(* CoDeSys 2.3.9.42 project: PROYECTO_FINAL.pro *)
(* Libraries: Standard.LIB 4.10.05 12:14:46, Iecsfc.lib 13.4.06 15:51:28 *)

(* Global variable list: Global_Variables *)
VAR_GLOBAL


(*ENTRADAS*)

	M:BOOL;(*Boton para iniciar el proceso automatico*)
	Marcha:BOOL;(*Variable que se pone a 1 cuando apretamos M*)
	Auto:BOOL;(*Cambio de modo automatico a manual*)


	P:BOOL;(*Boton para parar el proceso automatico*)
	E:BOOL;(*Boton para iniciar el proceso de emergencia*)
	Rearme:BOOL;(*Boton para reiniciar el proceso*)

	Mesa1:BOOL;(*Boton para Mesa 1*)
	Mesa2:BOOL;(*Boton para Mesa 2*)
	Mesa3:BOOL;(*Boton para Mesa 3*)
	Mesa4:BOOL;(*Boton para Mesa 4*)


	Pizza1:BOOL;(*Boton pizza 1: Tomate y queso*)
	Pizza2:BOOL;(*Boton pizza 2: Tomate, queso y jamon*)
	Pizza3:BOOL;(*Boton pizza 3:Tomate,queso y peperoni*)
	Pizza4:BOOL;(*Boton pizza 4:Tomate, queso, pimientos y champiñones*)
	P1:BOOL;(*Variable que se pone a 1 cuando se elige la pizza 1 y que se pone a 0 cuando se entra en el horno*)
	P2:BOOL;(*Variable que se pone a 1 cuando se elige la pizza 2 y que se pone a 0 cuando se entra en el horno*)
	P3:BOOL;(*Variable que se pone a 1 cuando se elige la pizza 3 y que se pone a 0 cuando se entra en el horno*)
	P4:BOOL;(*Variable que se pone a 1 cuando se elige la pizza 4 y que se pone a 0 cuando se entra en el horno*)


	SMasa:BOOL;(*Sensor de que la masa cae en la cinta*)
	SAmasador:BOOL;(*Sensor de que la masa esta en el punto de amasar*)

	(*Sensores ingredientes*)
	SPizza:BOOL;(*Sensor para ver que pizza se ha elegido*)
	STOM:BOOL;(*Sensor que la pizza esta en la posicion para echar tomate*)
	SQUE:BOOL;(*Sensor que la pizza esta en la posicion para echar queso*)
	SJAM:BOOL;(*Sensor que la pizza esta en la posicion para echar jamon*)
	SPEP: BOOL;(*Sensor que la pizza esta en la posicion para echar peperoni*)
	SPIM: BOOL;(*Sensor que la pizza esta en la posicion para echar pimiento*)
	SCHAMP: BOOL;(*Sensor que la pizza esta en la posicion para echar champiñones*)
	SHORNO: BOOL;(*Sensor que se activa cuando la pizza llega al horno*)
	SCarrito:BOOL;(*Sensor que se activa cuando hay un carrito en la salida del horno*)
	SMesa1:BOOL;(*Sensor que se activa cuando carrito llega a mesa 1*)
	SMesa2:BOOL;(*Sensor que se activa cuando carrito llega a mesa 2*)
	SMesa3:BOOL;(*Sensor que se activa cuando carrito llega a mesa 3*)
	SMesa4:BOOL;(*Sensor que se activa cuando carrito llega a mesa 4*)

	SEHorno:BOOL;(*Sensor de entrada horno*)
	SFHorno:BOOL;(*Sensor salida horno*)
	INVISIBLE:BOOL;(*Se activa para hacer invisible la masa*)

	(*Botones del modo Manual*)
	MAS:BOOL;(*Boton para tirar una masa a la cinta*)
	MOT:BOOL;(*Boton que activa la cinta*)
	AM:BOOL;(*Boton de amasar*)
	TOM:BOOL;(*Boton del tomate*)
	QUE:BOOL;(*Boton del queso*)
	JAM:BOOL;(*Boton del jamon*)
	PEP:BOOL;(*Boton del peperoni*)
	PIM:BOOL;(*Boton del pimiento*)
	CH:BOOL;(*Boton de los champiñones*)
	H:BOOL;(*Boton del horno*)

	(*posicion carrito*)
	PosYR:INT;(*Coordenada Y carrito*)
	PosXR:INT;(*Coordenada X carrito*)
	ActMesa1: BOOL;(*variable que se activa al elegir la mesa 1*)
	ActMesa2: BOOL;(*variable que se activa al elegir la mesa 2*)
	ActMesa3: BOOL;(*variable que se activa al elegir la mesa 3*)
	ActMesa4: BOOL;(*variable que se activa al elegir la mesa 4*)
	CargaRojo: BOOL;(*Variable para mostrar que la pizza se ha cargado en el carrito*)
	(*posicion masa*)
	PosXM:INT;
	PosYM:INT;
	AUXMasa:BOOL;(*variable auxiliar que se activa mientras la masa cae en la cinta*)





(*SALIDAS*)

	(*Acciones de la cinta*)
	Masa:BOOL;(*Accion de tirar la masa en la cinta*)
	Amasador:BOOL;(*Accion de amasar la masa*)
	Motor:BOOL;(*Motor de la cinta*)
	Horno:BOOL;(*Horno encendido*)

	(*Acciones ingredientes*)
	MT:BOOL;(*Abrir compuerta del tomate*)
	MQ:BOOL;(*Abrir compuerta del queso*)
	MJ:BOOL;(*Abrir compuerta del jamon*)
	MPE:BOOL;(*Abrir compuerta del peperoni*)
	MPI:BOOL;(*Abrir compuerta del pimiento*)
	MCH:BOOL;(*Abrir compuerta de los champiñones*)


	Vel:INT:=2;(*Velocidad para las animaciones*)






END_VAR

(* POU PLC_PRG, ST *)
PROGRAM PLC_PRG

VAR

END_VAR
Cinta;
Control;
Cambio_Modo;
Amasadora;
ControlCarritoRojo;
END_PROGRAM

(* POU CINTA_TRANSPORTADORA/Cinta, ST *)
PROGRAM Cinta
VAR

END_VAR
SMasa:=FALSE;
	SAmasador:=FALSE;
	SPizza:=FALSE;
	STOM:=FALSE;
	SQUE:=FALSE;
	SJAM:=FALSE;
	SPEP:=FALSE;
	SPIM:=FALSE;
	SCHAMP:=FALSE;
	SHORNO:=FALSE;
	SEHORNO:=FALSE;
	SFHORNO:=FALSE;

IF PosYM>=0 AND PosYM<=80 AND PosXM=0 THEN
AUXMasa:=TRUE;
END_IF


IF Masa=TRUE THEN
	PosYM:=PosYM+Vel;

END_IF

IF Motor=TRUE  THEN
	 PosXM:=PosXM+Vel;
END_IF





IF PosYM>=80AND PosXM >=0 AND PosXM<=30 THEN
	SMasa:=TRUE;
	END_IF
IF PosXM >=80 AND PosXM<=120 THEN
 SAmasador:=TRUE;
	END_IF
IF PosXM>=200 AND PosXM<=240 THEN
 SPizza:=TRUE;
	END_IF
IF PosXM >=300 AND PosXM<=340 THEN
 STOM:=TRUE;
	END_IF
IF PosXM>=370 AND PosXM<=390 THEN
 SQUE:=TRUE;
	END_IF
IF PosXM >=440 AND PosXM<=460 THEN
 SJAM:=TRUE;
	END_IF
IF PosXM >=510 AND PosXM<=530 THEN
 SPEP:=TRUE;
	END_IF
IF PosXM >=580 AND PosXM<=600 THEN
 SPIM:=TRUE;
	END_IF
IF PosXM >=650 AND PosXM<=670 THEN
 SCHAMP:=TRUE;
	END_IF
IF PosXM >=720 AND PosXM<=750 THEN
 SEHORNO:=TRUE;
	END_IF
IF PosXM >=820 AND PosXM<=840 THEN
 SFHORNO:=TRUE;
	END_IF
IF INVISIBLE=TRUE THEN
PosXM:=0;
PosYM:=0;
INVISIBLE:=FALSE;
END_IF

IF SMasa=TRUE THEN
AUXMasa:=FALSE;
END_IF
END_PROGRAM

(* POU CONTROL_AUTO/MAN/Control, SFC *)
PROGRAM Control
VAR
	OK:BOOL;
END_VAR
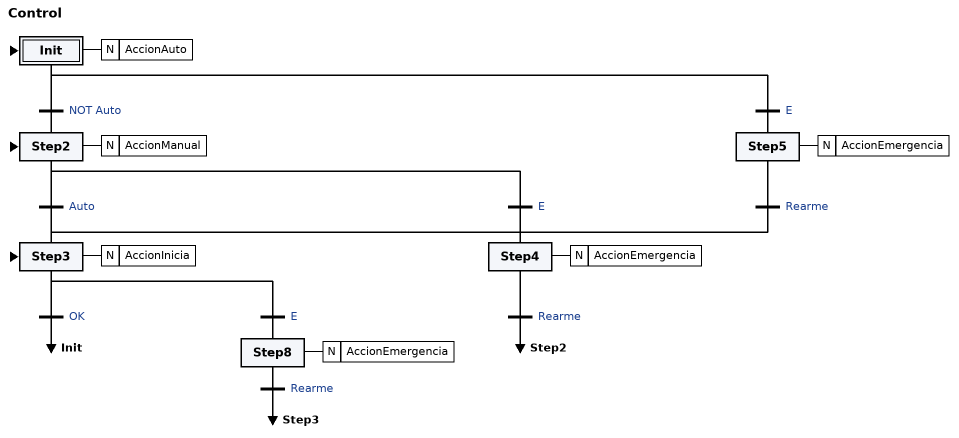
INITIAL_STEP Init:
	AccionAuto(N);
END_STEP
TRANSITION FROM Init TO Step2 := NOT Auto;
END_TRANSITION
TRANSITION FROM Init TO Step5 := E;
END_TRANSITION
STEP Step5:
	AccionEmergencia(N);
END_STEP
TRANSITION FROM Step5 TO Step3 := Rearme;
END_TRANSITION
STEP Step2:
	AccionManual(N);
END_STEP
TRANSITION FROM Step2 TO Step3 := Auto;
END_TRANSITION
TRANSITION FROM Step2 TO Step4 := E;
END_TRANSITION
STEP Step4:
	AccionEmergencia(N);
END_STEP
TRANSITION FROM Step4 TO Step2 := Rearme;
END_TRANSITION
STEP Step3:
	AccionInicia(N);
END_STEP
TRANSITION FROM Step3 TO Init := OK;
END_TRANSITION
TRANSITION FROM Step3 TO Step8 := E;
END_TRANSITION
STEP Step8:
	AccionEmergencia(N);
END_STEP
TRANSITION FROM Step8 TO Step3 := Rearme;
END_TRANSITION
END_PROGRAM
ACTION AccionAuto:
Cinta_Auto(SFCReset:=FALSE);

Arranque();
END_ACTION
ACTION AccionEmergencia:
PosXM:=0;
PosYM:=0;
PosYR:=0;
PosXR:=0;
MT:=FALSE;
Masa:=FALSE;
MQ:=FALSE;
MJ:=FALSE;
MPE:=FALSE;
MPI:=FALSE;
MCH:=FALSE;
Horno:=FALSE;
Amasador:=FALSE;
Marcha:=FALSE;
ActMesa1:=FALSE;
	ActMesa2:=FALSE;
	ActMesa3:=FALSE;
	ActMesa4:=FALSE;
CargaRojo:=FALSE;
END_ACTION
ACTION AccionInicia:
Cinta_Auto(SFCReset:=TRUE);
IF PosYM>=-2 AND PosYM<=2 AND PosXM>=-2 AND PosXM<=2 THEN
OK:=TRUE;
ELSE
OK:=FALSE;
END_IF
END_ACTION
ACTION AccionManual:
Cinta_Manual();
END_ACTION

(* POU CINTA_TRANSPORTADORA/Cinta_Auto, SFC *)
PROGRAM Cinta_Auto
VAR_INPUT
	SFCReset:BOOL;

END_VAR
VAR
	P1:BOOL;
	P2:BOOL;
	P3:BOOL;
	P4:BOOL;

END_VAR
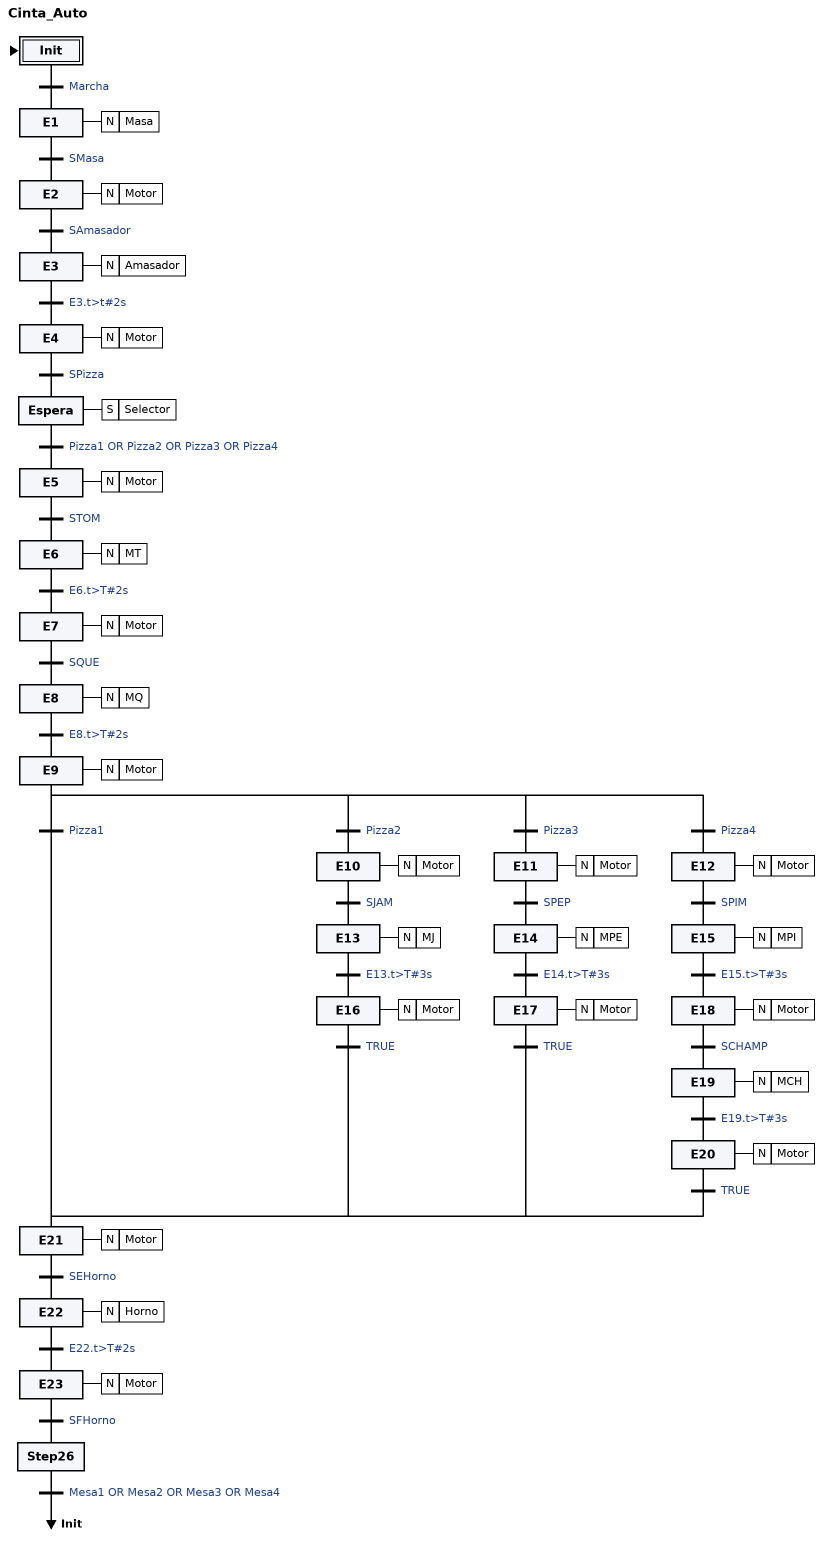
INITIAL_STEP Init:
END_STEP
TRANSITION FROM Init TO E1 := Marcha;
END_TRANSITION
STEP E1:
	Masa(N);
END_STEP
TRANSITION FROM E1 TO E2 := SMasa;
END_TRANSITION
STEP E2:
	Motor(N);
END_STEP
TRANSITION FROM E2 TO E3 := SAmasador;
END_TRANSITION
STEP E3:
	Amasador(N);
END_STEP
TRANSITION FROM E3 TO E4 := E3.t>t#2s;
END_TRANSITION
STEP E4:
	Motor(N);
END_STEP
TRANSITION FROM E4 TO Espera := SPizza;
END_TRANSITION
STEP Espera:
	Selector(S);
END_STEP
TRANSITION FROM Espera TO E5 := Pizza1 OR Pizza2 OR Pizza3 OR Pizza4;
END_TRANSITION
STEP E5:
	Motor(N);
END_STEP
TRANSITION FROM E5 TO E6 := STOM;
END_TRANSITION
STEP E6:
	MT(N);
END_STEP
TRANSITION FROM E6 TO E7 := E6.t>T#2s;
END_TRANSITION
STEP E7:
	Motor(N);
END_STEP
TRANSITION FROM E7 TO E8 := SQUE;
END_TRANSITION
STEP E8:
	MQ(N);
END_STEP
TRANSITION FROM E8 TO E9 := E8.t>T#2s;
END_TRANSITION
STEP E9:
	Motor(N);
END_STEP
TRANSITION FROM E9 TO E21 := Pizza1;
END_TRANSITION
TRANSITION FROM E9 TO E10 := Pizza2;
END_TRANSITION
TRANSITION FROM E9 TO E11 := Pizza3;
END_TRANSITION
TRANSITION FROM E9 TO E12 := Pizza4;
END_TRANSITION
STEP E10:
	Motor(N);
END_STEP
TRANSITION FROM E10 TO E13 := SJAM;
END_TRANSITION
STEP E13:
	MJ(N);
END_STEP
TRANSITION FROM E13 TO E16 := E13.t>T#3s;
END_TRANSITION
STEP E16:
	Motor(N);
END_STEP
TRANSITION FROM E16 TO E21 := TRUE;
END_TRANSITION
STEP E11:
	Motor(N);
END_STEP
TRANSITION FROM E11 TO E14 := SPEP;
END_TRANSITION
STEP E14:
	MPE(N);
END_STEP
TRANSITION FROM E14 TO E17 := E14.t>T#3s;
END_TRANSITION
STEP E17:
	Motor(N);
END_STEP
TRANSITION FROM E17 TO E21 := TRUE;
END_TRANSITION
STEP E12:
	Motor(N);
END_STEP
TRANSITION FROM E12 TO E15 := SPIM;
END_TRANSITION
STEP E15:
	MPI(N);
END_STEP
TRANSITION FROM E15 TO E18 := E15.t>T#3s;
END_TRANSITION
STEP E18:
	Motor(N);
END_STEP
TRANSITION FROM E18 TO E19 := SCHAMP;
END_TRANSITION
STEP E19:
	MCH(N);
END_STEP
TRANSITION FROM E19 TO E20 := E19.t>T#3s;
END_TRANSITION
STEP E20:
	Motor(N);
END_STEP
TRANSITION FROM E20 TO E21 := TRUE;
END_TRANSITION
STEP E21:
	Motor(N);
END_STEP
TRANSITION FROM E21 TO E22 := SEHorno;
END_TRANSITION
STEP E22:
	Horno(N);
END_STEP
TRANSITION FROM E22 TO E23 := E22.t>T#2s;
END_TRANSITION
STEP E23:
	Motor(N);
END_STEP
TRANSITION FROM E23 TO Step26 := SFHorno;
END_TRANSITION
STEP Step26:
END_STEP
TRANSITION FROM Step26 TO Init := Mesa1 OR Mesa2 OR Mesa3 OR Mesa4;
END_TRANSITION
END_PROGRAM
ACTION Selector:
Seleccion_Pizza();
END_ACTION

(* POU CINTA_TRANSPORTADORA/Seleccion_Pizza, ST *)
PROGRAM Seleccion_Pizza
VAR
END_VAR
IF P1=TRUE THEN
	Pizza1:=TRUE;
END_IF
IF P2=TRUE THEN
	Pizza2:=TRUE;
END_IF
IF P3=TRUE THEN
	Pizza3:=TRUE;
END_IF
IF P4=TRUE THEN
	Pizza4:=TRUE;
END_IF

IF Mesa1 OR Mesa2 OR Mesa3 OR MEsa4 THEN
Pizza1:=FALSE;
Pizza2:=FALSE;
Pizza3:=FALSE;
Pizza4:=FALSE;
END_IF
END_PROGRAM

(* POU CINTA_TRANSPORTADORA/Cinta_Manual, LD *)
PROGRAM Cinta_Manual
VAR
	Temp: TOF;

END_VAR
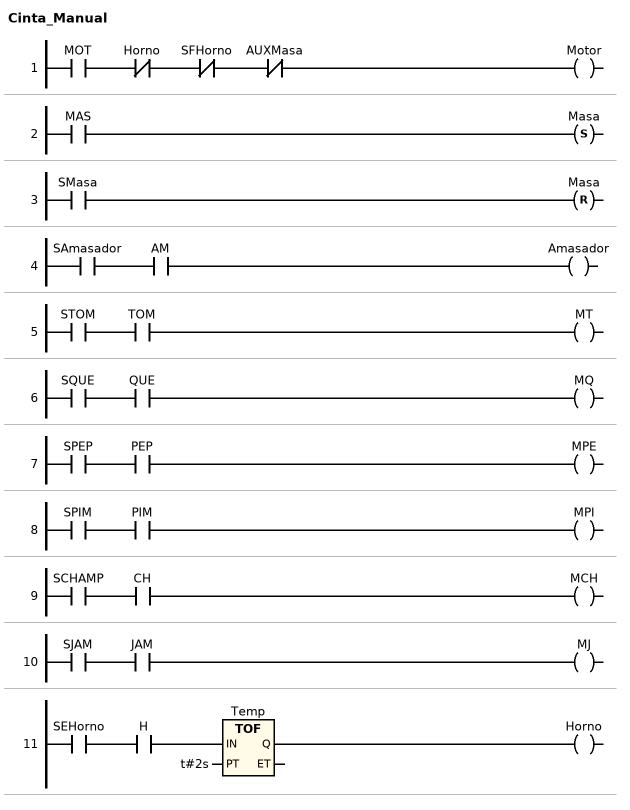
_LD_ (* Ladder Diagram *)
NETWORK 1
	[MOT] - [/Horno] - [/SFHorno] - [/AUXMasa] --- (Motor)
NETWORK 2
	[MAS] --- (S Masa)
NETWORK 3
	[SMasa] --- (R Masa)
NETWORK 4
	[SAmasador] - [AM] --- (Amasador)
NETWORK 5
	[STOM] - [TOM] --- (MT)
NETWORK 6
	[SQUE] - [QUE] --- (MQ)
NETWORK 7
	[SPEP] - [PEP] --- (MPE)
NETWORK 8
	[SPIM] - [PIM] --- (MPI)
NETWORK 9
	[SCHAMP] - [CH] --- (MCH)
NETWORK 10
	[SJAM] - [JAM] --- (MJ)
NETWORK 11
	[SEHorno] - [H] - Temp:TOF(IN: *, PT: t#2s) --- (Horno)
_END_LD_
(* the same logic as Structured Text *)
(* Network 1 *)
Motor := MOT AND NOT Horno AND NOT SFHorno AND NOT AUXMasa;
(* Network 2 *)
IF MAS THEN Masa := TRUE; END_IF;
(* Network 3 *)
IF SMasa THEN Masa := FALSE; END_IF;
(* Network 4 *)
Amasador := SAmasador AND AM;
(* Network 5 *)
MT := STOM AND TOM;
(* Network 6 *)
MQ := SQUE AND QUE;
(* Network 7 *)
MPE := SPEP AND PEP;
(* Network 8 *)
MPI := SPIM AND PIM;
(* Network 9 *)
MCH := SCHAMP AND CH;
(* Network 10 *)
MJ := SJAM AND JAM;
(* Network 11 *)
Temp(IN := SEHorno AND H, PT := t#2s);
Horno := Temp.Q;
END_PROGRAM

(* POU CONTROL_AUTO/MAN/Cambio_Modo, ST *)
PROGRAM Cambio_Modo
VAR
	Texto:STRING;
END_VAR
IF Auto THEN
  Texto:='Auto';
ELSE
   Texto:='Manual';
END_IF
END_PROGRAM

(* POU CINTA_TRANSPORTADORA/Amasadora, ST *)
PROGRAM Amasadora
VAR
	PosY:INT;
	aux:BOOL;
END_VAR
VAR_INPUT
END_VAR
IF Amasador=TRUE AND PosY<=60 THEN
PosY:=PosY+Vel;
aux:=TRUE;
END_IF


IF Amasador=FALSE AND aux=TRUE THEN
	PosY:=PosY-Vel;
END_IF

IF PosY= 0 THEN
	aux:=FALSE;
END_IF
END_PROGRAM

(* POU ControlCarritoRojo, ST *)
PROGRAM ControlCarritoRojo
VAR

	TempCarga: TON;(*Tiempo para cargar la pizza en la mesa*)
	FT2: BOOL;

	VuelveX1:BOOL;(*Vuelta del carrito de la mesa 1*)
	VuelveY2: BOOL;(*Vuelta del carrito de la mesa 2*)
	VuelveY3:BOOL;(*Vuelta del carrito de la mesa 3*)
	VuelveY4: BOOL;(*Vuelta del carrito de la mesa 4*)

	(*Variables auxiliares*)
	aux1:BOOL;
	aux2:BOOL;
	aux3:BOOL;
	aux4:BOOL;





END_VAR
TempCarga(IN:=aux1 OR aux2 OR aux3 OR aux4,PT:=T#2s,Q=>FT2);
SCarrito:=FALSE;
SMesa2:=FALSE;
SMesa1:=FALSE;
SMesa3:=FALSE;
SMesa4:=FALSE;

IF PosXR>=80 AND PosXR <=110 THEN
	SMesa1:=TRUE;
END_IF
IF PosYR>=100AND PosYR <=110 THEN
	SMesa2:=TRUE;
END_IF
IF PosYR>=170 AND PosYR <=180 THEN
	SMesa3:=TRUE;
END_IF
IF PosYR>=250 AND PosYR <=260 THEN
	SMesa4:=TRUE;
END_IF



IF PosYR>=-5 AND PosYR<=5 AND PosXR>=-5 AND PosXR<=5 THEN
	SCarrito:=TRUE;
END_IF



IF SFHORNO=TRUE AND SCarrito AND( Mesa1 OR Mesa2 OR Mesa3 OR Mesa4) THEN
	CargaRojo:=TRUE;
	INVISIBLE:=TRUE;

END_IF

IF Mesa1=TRUE AND  SFHORNO=TRUE THEN
ActMesa1:=TRUE;
END_IF

IF Mesa2=TRUE AND SFHORNO=TRUE THEN
ActMesa2:=TRUE;
END_IF
IF Mesa3=TRUE AND SFHORNO=TRUE THEN
ActMesa3:=TRUE;
END_IF
IF Mesa4=TRUE AND SFHORNO=TRUE THEN
ActMesa4:=TRUE;
END_IF



(*Para la mesa1*)

IF ActMesa1=TRUE AND CargaRojo=TRUE THEN
	PosXR:=PosXR+Vel;
END_IF

IF SMesa1=TRUE THEN
	ActMesa1:=FALSE;
	aux1:=TRUE;
END_IF

IF FT2=TRUE AND SMesa1=TRUE THEN
VuelveX1:=TRUE;
END_IF


IF VuelveX1=TRUE THEN
	PosXR:=PosXR-Vel;
aux1:=FALSE;
CargaRojo:=FALSE;
END_IF


IF SCarrito=TRUE THEN
	VuelveX1:=FALSE;
END_IF



(*Para la mesa2*)
IF ActMesa2=TRUE AND CargaRojo=TRUE THEN
	PosYR:=PosYR+Vel;
END_IF

IF SMesa2=TRUE AND ActMesa2=TRUE THEN
	ActMesa2:=FALSE;
	aux2:=TRUE;
END_IF


IF FT2=TRUE  AND SMesa2=TRUE THEN
VuelveY2:=TRUE;
END_IF


IF VuelveY2=TRUE  THEN
	PosYR:=PosYR-Vel;
aux2:=FALSE;
CargaRojo:=FALSE;
END_IF


IF SCarrito=TRUE THEN
	VuelveY2:=FALSE;
END_IF

(*Para la mesa3*)
IF ActMesa3=TRUE AND CargaRojo=TRUE THEN
	PosYR:=PosYR+Vel;
END_IF

IF SMesa3=TRUE AND ActMesa3=TRUE THEN
	ActMesa3:=FALSE;
	aux3:=TRUE;
END_IF


IF FT2=TRUE  AND SMesa3=TRUE THEN
VuelveY3:=TRUE;
END_IF

IF VuelveY3=TRUE  THEN
	PosYR:=PosYR-Vel;
aux3:=FALSE;
CargaRojo:=FALSE;
END_IF


IF SCarrito=TRUE THEN
	VuelveY3:=FALSE;
END_IF

(*Para la mesa4*)
IF ActMesa4=TRUE AND CargaRojo=TRUE THEN
	PosYR:=PosYR+Vel;
END_IF

IF SMesa4=TRUE AND ActMesa4=TRUE THEN
	ActMesa4:=FALSE;
	aux4:=TRUE;
END_IF


IF FT2=TRUE AND SMesa4=TRUE THEN
 VuelveY4:=TRUE;
END_IF

IF VuelveY4=TRUE THEN
	PosYR:=PosYR-Vel;
aux4:=FALSE;
CargaRojo:=FALSE;
END_IF


IF SCarrito=TRUE THEN
	VuelveY4:=FALSE;
END_IF
END_PROGRAM

(* POU CONTROL_AUTO/MAN/Arranque, LD *)
PROGRAM Arranque
VAR
END_VAR
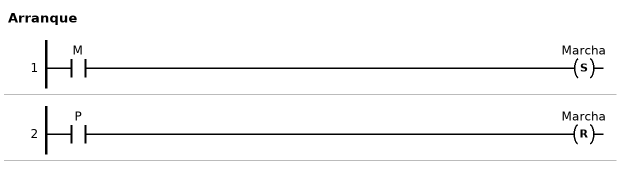
_LD_ (* Ladder Diagram *)
NETWORK 1
	[M] --- (S Marcha)
NETWORK 2
	[P] --- (R Marcha)
_END_LD_
(* the same logic as Structured Text *)
(* Network 1 *)
IF M THEN Marcha := TRUE; END_IF;
(* Network 2 *)
IF P THEN Marcha := FALSE; END_IF;
END_PROGRAM

(* Visualisation Sala_Pizzeria
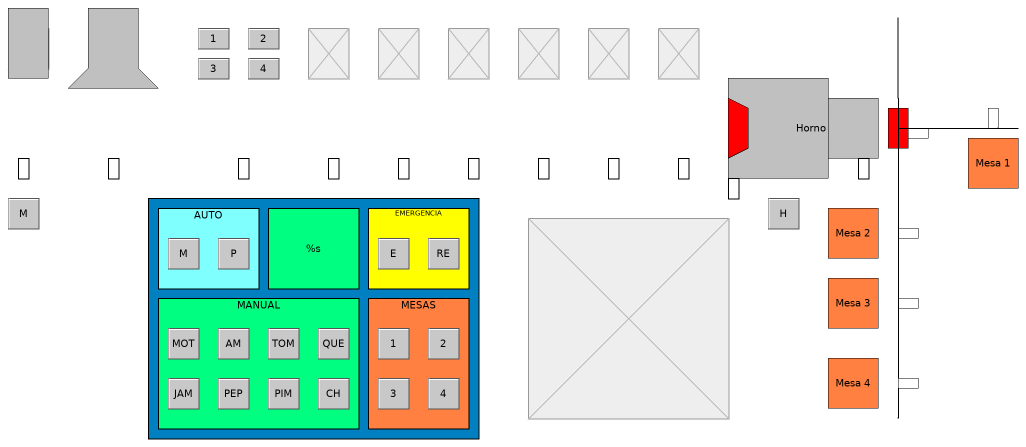
button at (240,60)-(271,81): text "1"; taps P1
button at (290,60)-(321,81): text "2"; taps P2
button at (240,90)-(271,111): text "3"; taps P3
button at (290,90)-(321,111): text "4"; taps P4
polygon at (870,390)-(920,440): text "Mesa 4"
rectangle at (150,190)-(161,211): alarm colour if SAmasador; toggles SAmasador
rectangle at (60,190)-(71,211): alarm colour if SMasa
rectangle at (280,190)-(291,211): alarm colour if SPizza
rectangle at (370,190)-(381,211): alarm colour if STOM
rectangle at (440,190)-(451,211): alarm colour if SQUE
rectangle at (510,190)-(521,211): alarm colour if SJAM
rectangle at (580,190)-(591,211): alarm colour if SPEP
rectangle at (650,190)-(661,211): alarm colour if SPIM
rectangle at (720,190)-(731,211): alarm colour if SCHAMP
rectangle at (310,240)-(401,321): text "%s"; shows CAMBIO_MODO.Texto; alarm colour if Auto; toggles Auto
rectangle at (770,210)-(781,231): alarm colour if SEHORNO
rectangle at (900,190)-(911,211): alarm colour if SFHORNO
polygon at (930,140)-(950,180): alarm colour if CargaRojo; x offset PosXR; y offset PosYR
polygon at (950,160)-(970,170): alarm colour if SCarrito
polygon at (1030,140)-(1040,160): alarm colour if SMesa1
polygon at (940,330)-(960,340): alarm colour if SMesa3
polygon at (940,260)-(960,270): alarm colour if SMesa2
polygon at (1010,170)-(1060,220): text "Mesa 1"
polygon at (870,240)-(920,290): text "Mesa 2"
polygon at (870,310)-(920,360): text "Mesa 3"
rectangle at (410,330)-(511,461): text "MESAS"
button at (420,360)-(451,391): text "1"; taps Mesa1
button at (470,360)-(501,391): text "2"; taps Mesa2
button at (470,410)-(501,441): text "4"; taps Mesa4
button at (420,410)-(451,441): text "3"; taps Mesa3
rectangle at (200,240)-(301,321): text "AUTO"
button at (210,270)-(241,301): text "M"; taps M
button at (260,270)-(291,301): text "P"; taps P
rectangle at (200,330)-(401,461): text "MANUAL"
button at (210,360)-(241,391): text "MOT"; toggles MOT; taps MOT
button at (310,360)-(341,391): text "TOM"; taps TOM
button at (260,410)-(291,441): text "PEP"; taps PEP
button at (360,360)-(391,391): text "QUE"; taps QUE
button at (310,410)-(341,441): text "PIM"; taps PIM
button at (360,410)-(391,441): text "CH"; taps CH
button at (260,360)-(291,391): text "AM"; taps AM
button at (210,410)-(241,441): text "JAM"; taps JAM
rectangle at (410,240)-(511,321): text "EMERGENCIA"
bitmap at (350,60)-(391,111): c:\users\aleja\onedrive\escritorio\alejandro uni\2º\automatización\proyecto\imagenes\tomate2.bmp
bitmap at (420,60)-(461,111): c:\users\aleja\onedrive\escritorio\alejandro uni\2º\automatización\proyecto\imagenes\queso2.bmp
bitmap at (490,60)-(531,111): c:\users\aleja\onedrive\escritorio\alejandro uni\2º\automatización\proyecto\imagenes\jamon-york.bmp
bitmap at (560,60)-(601,111): c:\users\aleja\onedrive\escritorio\alejandro uni\2º\automatización\proyecto\imagenes\peperoni.bmp
bitmap at (630,60)-(671,111): c:\users\aleja\onedrive\escritorio\alejandro uni\2º\automatización\proyecto\imagenes\pimverde.bmp
bitmap at (700,60)-(741,111): c:\users\aleja\onedrive\escritorio\alejandro uni\2º\automatización\proyecto\imagenes\champ.bmp
button at (810,230)-(841,261): text "H"; taps H
button at (420,270)-(451,301): text "E"; taps E
button at (470,270)-(501,301): text "RE"; taps Rearme
polygon at (940,410)-(960,420): alarm colour if SMesa4
bitmap at (570,250)-(771,451): pizza-logo-design-template-vector-png.bmp
button at (50,230)-(81,261): text "M"; taps MAS
bitmap at (50,60)-(91,101): c:\users\aleja\onedrive\escritorio\alejandro uni\2º\automatización\proyecto\masa.bmp
polygon at (110,40)-(200,120): y offset Amasadora.PosY
polygon at (770,110)-(870,210): text "Horno"
polygon at (770,130)-(790,190): alarm colour if Horno
6 more shapes without text or variables
1 elements of other kinds (tables, trends, ...) not read
*)
